// TIA Portal V19 export
ORGANIZATION_BLOCK "Main"   // OB1, LAD, ProgramCycle
TITLE = "Main Program Sweep (Cycle)"
{ S7_Optimized_Access := 'TRUE' }
// stored: SetENOAutomatically false
   VAR_INPUT
      Initial_Call : Bool;   // Initial call of this OB
      Remanence : Bool;   // =True, if remanent data are available
   END_VAR
BEGIN

REGION Network 1: Write clockbyte out to RH System, Display RH System clock byte inline
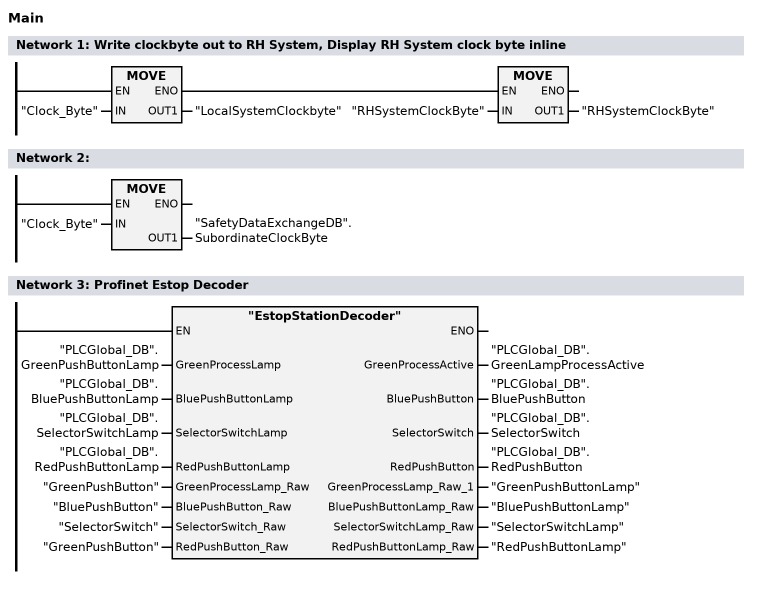
   RUNG wire#powerrail
      Move(in := "Clock_Byte", out1 => "LocalSystemClockbyte")
      Move(in := "RHSystemClockByte", out1 => "RHSystemClockByte")
   END_RUNG
   // the same network as SCL:
   "LocalSystemClockbyte" := "Clock_Byte";
   "RHSystemClockByte" := "RHSystemClockByte";
END_REGION

REGION Network 2
   RUNG wire#powerrail
      Move(in := "Clock_Byte", out1 => "SafetyDataExchangeDB".SubordinateClockByte)
   END_RUNG
   // the same network as SCL:
   "SafetyDataExchangeDB".SubordinateClockByte := "Clock_Byte";
END_REGION

REGION Network 3: Profinet Estop Decoder
   RUNG wire#powerrail
      "EstopStationDecoder"(GreenProcessLamp := "PLCGlobal_DB".GreenPushButtonLamp, BluePushButtonLamp := "PLCGlobal_DB".BluePushButtonLamp, SelectorSwitchLamp := "PLCGlobal_DB".SelectorSwitchLamp, RedPushButtonLamp := "PLCGlobal_DB".RedPushButtonLamp, GreenProcessLamp_Raw := "GreenPushButton", BluePushButton_Raw := "BluePushButton", SelectorSwitch_Raw := "SelectorSwitch", RedPushButton_Raw := "GreenPushButton", GreenProcessActive => "PLCGlobal_DB".GreenLampProcessActive, BluePushButton => "PLCGlobal_DB".BluePushButton, SelectorSwitch => "PLCGlobal_DB".SelectorSwitch, RedPushButton => "PLCGlobal_DB".RedPushButton, GreenProcessLamp_Raw_1 => "GreenPushButtonLamp", BluePushButtonLamp_Raw => "BluePushButtonLamp", SelectorSwitchLamp_Raw => "SelectorSwitchLamp", RedPushButtonLamp_Raw => "RedPushButtonLamp")
   END_RUNG
   // the same network as SCL:
   "EstopStationDecoder"(GreenProcessLamp := "PLCGlobal_DB".GreenPushButtonLamp,
                         BluePushButtonLamp := "PLCGlobal_DB".BluePushButtonLamp,
                         SelectorSwitchLamp := "PLCGlobal_DB".SelectorSwitchLamp,
                         RedPushButtonLamp := "PLCGlobal_DB".RedPushButtonLamp,
                         GreenProcessLamp_Raw := "GreenPushButton",
                         BluePushButton_Raw := "BluePushButton",
                         SelectorSwitch_Raw := "SelectorSwitch",
                         RedPushButton_Raw := "GreenPushButton",
                         GreenProcessActive => "PLCGlobal_DB".GreenLampProcessActive,
                         BluePushButton => "PLCGlobal_DB".BluePushButton,
                         SelectorSwitch => "PLCGlobal_DB".SelectorSwitch,
                         RedPushButton => "PLCGlobal_DB".RedPushButton,
                         GreenProcessLamp_Raw_1 => "GreenPushButtonLamp",
                         BluePushButtonLamp_Raw => "BluePushButtonLamp",
                         SelectorSwitchLamp_Raw => "SelectorSwitchLamp",
                         RedPushButtonLamp_Raw => "RedPushButtonLamp");
END_REGION
END_ORGANIZATION_BLOCK
